FUNCTION_BLOCK FB_TrackSegment_3 EXTENDS FB_TrackBase IMPLEMENTS I_TRACK
VAR_INPUT
END_VAR
VAR_OUTPUT
END_VAR

METHOD Initialize : BOOL

VAR_INPUT
	nTrackIndex : UDINT;
END_VAR


VAR_INST
	TrackTable		: FB_TrackTable;
	
	nPointIndex		: INT;
	nPointIndexA	: INT;	
	nPointIndexB	: INT;	
	idx1, idx2		: INT;
	nStartFromTrack	: INT;
	nEndAtTrack		: INT;
	bCloseLoop		: BOOL;	
	
	bTrackBuild		: BOOL;
	StartFromTrack	: I_Track;
	EndAtTrack		: I_Track;
	
	sIndexWhereTheCheckFailed	: UINT;
	nErrorID					: UDINT;

END_VAR





VAR_INST
	
	TrackTableTemp		: ARRAY[1..gc_MaxNumberTrackPoints] OF ST_TrackTable;
	


END_VAR


VAR_INST
	
	pos01	:		PositionXYC;
	pos02	:		PositionXYC;


END_VAR

	  
CASE nState OF 

	10:	// Starting with an empty table. 
		IF TrackTable.ClearTrackTable() THEN
			nState := nState + 10;
		END_IF
		

	20:	// Init Track-Table
		
		// *************************************************************************************
		// *** Only the code in this state must be eddited according to machine/track layout ***
		// *************************************************************************************	
		
		nStartFromTrack	:= 1;		// 0 for the first track all others according to their predecessor!
	    	nEndAtTrack := 1;		// 0 for the first track all others according to their successor! 		
		     bCloseLoop := FALSE;	// TRUE for circular track	

			 			 			 
		// Building the track table:
		TrackTable.AddPoint(E_PointType.Line_Start, E_PointOption.none, 480.0, 600.0, 0.0); 	 
		TrackTable.AddPoint(E_PointType.Line_End,   E_PointOption.none, 720.0, 600.0, 0.0);				
						
		TrackTable.AddPoint(E_PointType.Line_Start, E_PointOption.none, 840.0, 480.0, 0.0); 	 
		TrackTable.AddPoint(E_PointType.Line_End,   E_PointOption.none, 840.0, 240.0, 0.0);			
		
		TrackTable.AddPoint(E_PointType.Line_Start, E_PointOption.none, 720.0, 120.0, 0.0); 	 
		TrackTable.AddPoint(E_PointType.Line_End,   E_PointOption.none, 480.0, 120.0, 0.0);			
		
		nState := nState + 10;

		
	30:
		// *************************************************************
		// ***       NO Code Changes are needed from here on!        ***
		// *************************************************************		
			
		// The track table contains all additional information, too.
		IF nStartFromTrack > 0 THEN
			TrackTable.P_StartFromTrack := ipTrack[nStartFromTrack].std;	
		END_IF
		IF nEndAtTrack > 0 THEN
			TrackTable.P_EndAtTrack := ipTrack[nEndAtTrack].std;	
		END_IF	
		TrackTable.P_CloseTheLoop := bCloseLoop;	
		nState := nState + 10;

			
		
	40: // Checking the track table for plausibility
		IF TrackTable.CheckTrackTable() <> 0 THEN
			IF TrackTable.P_TrackTableCheckResult THEN
				nState := 50;	// Plausibility test succeeded.
			ELSE
				nState := 41;	// Plausibility test failed!
			END_IF
		END_IF

	
	41:	// In case of failed plausibility test check the creation of the above track table.
		// A Line must always begin with E_PointType.Line_Start and end with E_PointType.Line_End.
		// A Circle must always be added in the order E_PointType.Circle_Start, E_PointType.Circle_Center, E_PointType.Circle_End.
		// Check the info text for further information:
		sErrorInfoTextTemp := CONCAT('Track: ', UDINT_TO_STRING(nTrackIndex));
		sErrorInfoTextTemp := CONCAT(sErrorInfoTextTemp, ' - ');
		sErrorInfoTextTemp := CONCAT(sErrorInfoTextTemp, TrackTable.P_InfoText);
		
				     bTrackBuildError := TRUE;
					   sErrorInfoText := sErrorInfoTextTemp;
			sIndexWhereTheCheckFailed := TrackTable.P_TrackCheckImplausibleTableIndex;
					   TrackTableTemp := TrackTable.P_Table;	
							
 					   
	50:	// Building the track	
		IF fbTrackStandard.BuildTrackExt(TrackTable) THEN
			nState := nState +1;
		END_IF
		
	51:	IF fbTrackStandard.P_BuildTrackExt.Done THEN
			nState := 100;	
		ELSIF fbTrackStandard.P_BuildTrackExt.Error THEN
	  		nState := nState +1;
		END_IF		
		
	52: // In case an error occured, check the error ID and InfoText and react accordingly:
		sErrorInfoTextTemp := CONCAT('Track: ', UDINT_TO_STRING(nTrackIndex));
		sErrorInfoTextTemp := CONCAT(sErrorInfoTextTemp, ' - ');
		sErrorInfoTextTemp := CONCAT(sErrorInfoTextTemp, fbTrackStandard.P_BuildTrackExtInfoText);	
	
			      nErrorID := fbTrackStandard.P_BuildTrackExt.ErrorID;
		    sErrorInfoText := sErrorInfoTextTemp;		
			
		  bTrackBuildError := TRUE;		   
					   
		 
	100: 	// Track build done
			fTrackLength := fbTrackStandard.GetLength();
			  Initialize := TRUE;
	
			
END_CASE
END_METHOD

METHOD Initialize_Test : BOOL


VAR_INST
	TrackTable		: FB_TrackTable;
	
	nPointIndex		: INT;
	nPointIndexA	: INT;	
	nPointIndexB	: INT;	
	idx1, idx2		: INT;
	nStartFromTrack	: INT;
	nEndAtTrack		: INT;
	bCloseLoop		: BOOL;	
	
	bTrackBuild		: BOOL;
	StartFromTrack	: I_Track;
	EndAtTrack		: I_Track;
	
	sIndexWhereTheCheckFailed	: UINT;
	nErrorID					: UDINT;

END_VAR





VAR_INST
	
	TrackTableTemp		: ARRAY[1..maxNumTrackPoints] OF ST_TrackTable;
	


END_VAR


VAR_INST
	
	pos01	:		PositionXYC;
	pos02	:		PositionXYC;


END_VAR

	  
CASE nState OF 

	10:	// Starting with an empty table. 
		IF TrackTable.ClearTrackTable() THEN
			nState := nState + 10;
		END_IF
		

	20:	// Init Track-Table
		
		// *************************************************************************************
		// *** Only the code in this state must be eddited according to machine/track layout ***
		// *************************************************************************************	
		
		nStartFromTrack	:= 0;		// 0 for the first track all others according to their predecessor!
	    	nEndAtTrack := 0;		// 0 for the first track all others according to their successor! 		
		     bCloseLoop := TRUE;	// TRUE for circular track	

			 			 			 
		// Building the track table:
		TrackTable.AddPoint(E_PointType.Point, E_PointOption.none, 485.0, 605.0, 0.0); 	 
								
		TrackTable.AddPoint(E_PointType.Line_Start, E_PointOption.none, 490.0, 610.0, 0.0); 	 
		TrackTable.AddPoint(E_PointType.Line_End,   E_PointOption.none, 590.0, 690.0, 0.0);			
		 
		TrackTable.AddPoint(E_PointType.Circle_Start,  E_PointOption.none, 700.0, 700.0, 0.0);
		TrackTable.AddPoint(E_PointType.Circle_Center, E_PointOption.none, 700.0, 800.0, 0.0); 	 
		TrackTable.AddPoint(E_PointType.Circle_End,    E_PointOption.none, 700.0, 900.0, 0.0);			
		
		nState := nState + 10;

		
	30:
		// *************************************************************
		// ***       NO Code Changes are needed from here on!        ***
		// *************************************************************		
			
		// The track table contains all additional information, too.
		IF nStartFromTrack > 0 THEN
			TrackTable.P_StartFromTrack := ipTrack[nStartFromTrack].std;	
		END_IF
		IF nEndAtTrack > 0 THEN
			TrackTable.P_EndAtTrack := ipTrack[nEndAtTrack].std;	
		END_IF	
		TrackTable.P_CloseTheLoop := bCloseLoop;	
		nState := nState + 10;

			
		
	40: // Checking the track table for plausibility
		IF TrackTable.CheckTrackTable() <> 0 THEN
			IF TrackTable.P_TrackTableCheckResult THEN
				nState := 50;	// Plausibility test succeeded.
			ELSE
				nState := 41;	// Plausibility test failed!
			END_IF
		END_IF

	
	41:	// In case of failed plausibility test check the creation of the above track table.
		// A Line must always begin with E_PointType.Line_Start and end with E_PointType.Line_End.
		// A Circle must always be added in the order E_PointType.Circle_Start, E_PointType.Circle_Center, E_PointType.Circle_End.
		// Check the info text for further information:
				     bTrackBuildError := TRUE;
			           sErrorInfoText := TrackTable.P_InfoText;
			sIndexWhereTheCheckFailed := TrackTable.P_TrackCheckImplausibleTableIndex;
					   TrackTableTemp := TrackTable.P_Table;	
							
 			
	50:	// Building the track	
		IF fbTrackStandard.BuildTrackExt(TrackTable) THEN
			nState := nState +1;
		END_IF
		
	51:	IF fbTrackStandard.P_BuildTrackExt.Done THEN
			nState := 100;	
		ELSIF fbTrackStandard.P_BuildTrackExt.Error THEN
	  		nState := nState +1;
		END_IF		
		
	52: // In case an error occured, check the error ID and InfoText and react accordingly:
			      nErrorID := fbTrackStandard.P_BuildTrackExt.ErrorID;
		    sErrorInfoText := fbTrackStandard.P_BuildTrackExtInfoText;		
			
		  bTrackBuildError := TRUE;		   
					   
		 
	100: 	// Track build done
			fTrackLength := fbTrackStandard.GetLength();
			  Initialize := TRUE;
	
			
END_CASE
END_METHOD

PROPERTY P_Error : BOOL
GET
P_Error := bTrackBuildError;
END_GET
END_PROPERTY

PROPERTY P_ErrorInfo : STRING
GET
P_ErrorInfo := sErrorInfoText;
END_GET
END_PROPERTY

END_FUNCTION_BLOCK

(* stored: Version 1.1.0.1, ProductVersion 3.1.4024.13
   POU FB_TrackSegment_3: Id {b135ed43-8901-453d-92d2-c891bb598a7a}, SpecialFunc None
   Method Initialize: Id {70d5fcbf-59f0-447e-b3a7-5b559f3f2249}
   Method Initialize_Test: Id {09a20b62-0faf-4a8f-ab58-06b1c87c084e}
   Property P_Error: Id {b5cb092c-9afd-4036-8b80-c1535d98e03a}
   Get Get: Id {a12efd32-8aa1-495a-ac37-838a963907ca}
   Property P_ErrorInfo: Id {9d0e43b0-c3fe-47b0-84f5-b5b79c34a75b}
   Get Get: Id {2cd44448-c78a-48be-a42e-426eb3f68e32} *)
